(* CoDeSys 2.3.5.6 project: lyjak_03.pro *)
(* Libraries: Standard.lib*4.1.15 17:23:13, SYSLIBCALLBACK.LIB*4.1.15 17:23:13 *)

(* PLC configuration (modules and I/O channels)
Configuration EC4P-200 [Root] node -1, in %IB0 out %QB0 {EC4P_RestartPwrOn = WARMSTART; EC4P_MaxCycleTime = 20; EC4P_Com1BaudRate = 38400; EC4P_CAN1BaudRate = 125KBaud; EC4P_RoutingId = 127; EC4P_EasyNetId = 1; EC4P_EasyNetCfg = 0; EC4P_EasyNetCycleTime = 50; EC4P_RoutingChannel = CAN1; EC4P_IPFlags = 0; EC4P_IPAddress = 0; EC4P_SubNetMask = 0; EC4P_DefaultGateway = 0; EC4P_SummerWinterFlags = 0; EC4P_SummerWinterRule1 = 0; EC4P_SummerWinterRule2 = 0}
  Local I/O [EC4P_LocalIO] node 0, in %IB0 out %QB0 {EC4P_LocalInt = 0}
    I1 AT %IX0.0 [LocalBitInput] Input I1
    I2 AT %IX0.1 [LocalBitInput] Input I2
    I3 AT %IX0.2 [LocalBitInput] Input I3
    I4 AT %IX0.3 [LocalBitInput] Input I4
    I5 AT %IX0.4 [LocalBitInput] Input I5
    I6 AT %IX0.5 [LocalBitInput] Input I6
    I7 AT %IX0.6 [LocalBitInput] Input I7
    I8 AT %IX0.7 [LocalBitInput] Input I8
    I9 AT %IX1.0 [LocalBitInput] Input I9
    I10 AT %IX1.1 [LocalBitInput] Input I10
    I11 AT %IX1.2 [LocalBitInput] Input I11
    I12 AT %IX1.3 [LocalBitInput] Input I12
    I13 AT %IX1.4 [LocalDiagInput] Diagnostic Input I13
    I14 AT %IX1.5 [LocalDiagInput] Diagnostic Input I14
    I15 AT %IX1.6 [LocalDiagInput] Diagnostic Input I15
    I16 AT %IX1.7 [LocalDiagInput] Diagnostic Input I16
    I7_Analog AT %IW2 [LocalAnalogIn] Input I7, 10Bit, 0-10VDC
    I8_Analog AT %IW4 [LocalAnalogIn] Input I8, 10Bit, 0-10VDC
    I11_Analog AT %IW6 [LocalAnalogIn] Input I11, 10Bit, 0-10VDC
    I12_Analog AT %IW8 [LocalAnalogIn] Input I12, 10Bit, 0-10VDC
    Transistor Outputs [EC4P_TOutputs] node 0, in %IB10 out %QB0
      Q1 AT %QX0.0 [LocalBitOutput] Transistor-Output Q1
      Q2 AT %QX0.1 [LocalBitOutput] Transistor-Output Q2
      Q3 AT %QX0.2 [LocalBitOutput] Transistor-Output Q3
      Q4 AT %QX0.3 [LocalBitOutput] Transistor-Output Q4
      Q5 AT %QX0.4 [LocalBitOutput] Transistor-Output Q5
      Q6 AT %QX0.5 [LocalBitOutput] Transistor-Output Q6
      Q7 AT %QX0.6 [LocalBitOutput] Transistor-Output Q7
      Q8 AT %QX0.7 [LocalBitOutput] Transistor-Output Q8
    No Analog Output [EC4P_NoAnalogOutput] node 1, in %IB10 out %QB1
    No Keys [EC4P_NoKeys] node 2, in %IB10 out %QB1
    No Counter [EC4P_NoCounter] node 3, in %IB10 out %QB1
  Extension [EC4P_Extension] node 1, in %IB10 out %QB1
    No Extension [EC4P_NoExtension] node 0, in %IB10 out %QB1
*)

(* POU PLC_PRG, LD *)
PROGRAM PLC_PRG
VAR
	TON1: TON;
	CZAS1: TIME;
	F_TRIG1: F_TRIG;
	CZAS2: TIME;
	CZAS3: TIME;
	TON2: TON;
	Y1: BOOL;
	RESET: BOOL;
	TP1: TP;
	TP2: TP;
	TP_GEN: TP;
	CTU1: CTU;
	LICZBA: INT;
	R_TRIG1: R_TRIG;
	CTUD1: CTUD;
	D1: BOOL;
	LICZBA1: INT;
	UP_END: BOOL;
	GEN: BOOL;
	X1: BOOL;
	DF: R_TRIG;
	X3: BOOL;
	X4: BOOL;
	TP3: TP;
	CZAS11: TIME;
	TON3: TON;
	SW: BOOL;
	TON4: TON;
	TP52: TP;
	R_TRIG_GEN: R_TRIG;
	TON7: TON;
	CZAS7: TIME;
	W1: BOOL;
	TON_2: TON;
	FTRIG6: F_TRIG;
END_VAR
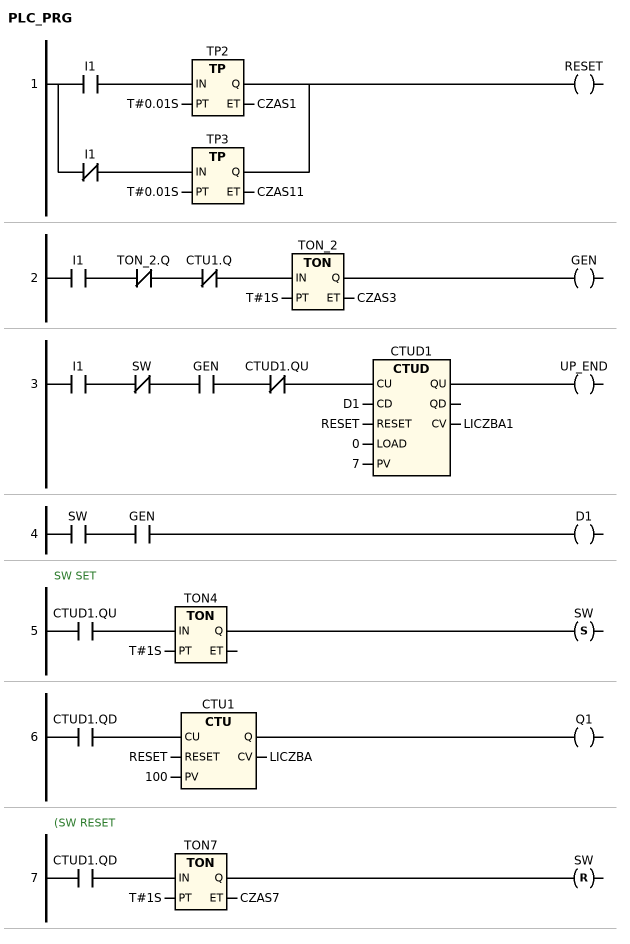
_LD_ (* Ladder Diagram *)
NETWORK 1
	{ [I1] - TP2:TP(IN: *, PT: T#0.01S, ET => CZAS1) | [/I1] - TP3:TP(IN: *, PT: T#0.01S, ET => CZAS11) } --- (RESET)
NETWORK 2
	[I1] - [/TON_2.Q] - [/CTU1.Q] - TON_2:TON(IN: *, PT: T#1S, ET => CZAS3) --- (GEN)
NETWORK 3
	[I1] - [/SW] - [GEN] - [/CTUD1.QU] - CTUD1:CTUD(CU: *, CD: D1, RESET: RESET, LOAD: 0, PV: 7, CV => LICZBA1) --- (UP_END)
NETWORK 4
	[SW] - [GEN] --- (D1)
NETWORK 5 (* SW SET *)
	[CTUD1.QU] - TON4:TON(IN: *, PT: T#1S) --- (S SW)
NETWORK 6
	[CTUD1.QD] - CTU1:CTU(CU: *, RESET: RESET, PV: 100, CV => LICZBA) --- (Q1)
NETWORK 7 (* (SW RESET *)
	[CTUD1.QD] - TON7:TON(IN: *, PT: T#1S, ET => CZAS7) --- (R SW)
_END_LD_
(* the same logic as Structured Text *)
(* Network 1 *)
TP2(IN := I1, PT := T#0.01S);
CZAS1 := TP2.ET;
TP3(IN := NOT I1, PT := T#0.01S);
CZAS11 := TP3.ET;
RESET := TP2.Q OR TP3.Q;
(* Network 2 *)
TON_2(IN := I1 AND NOT TON_2.Q AND NOT CTU1.Q, PT := T#1S);
CZAS3 := TON_2.ET;
GEN := TON_2.Q;
(* Network 3 *)
CTUD1(CU := I1 AND NOT SW AND GEN AND NOT CTUD1.QU, CD := D1, RESET := RESET, LOAD := 0, PV := 7);
LICZBA1 := CTUD1.CV;
UP_END := CTUD1.QU;
(* Network 4 *)
D1 := SW AND GEN;
(* Network 5: SW SET *)
TON4(IN := CTUD1.QU, PT := T#1S);
IF TON4.Q THEN SW := TRUE; END_IF;
(* Network 6 *)
CTU1(CU := CTUD1.QD, RESET := RESET, PV := 100);
LICZBA := CTU1.CV;
Q1 := CTU1.Q;
(* Network 7: (SW RESET *)
TON7(IN := CTUD1.QD, PT := T#1S);
CZAS7 := TON7.ET;
IF TON7.Q THEN SW := FALSE; END_IF;
END_PROGRAM
